CODESYSSPV3/3S/IecVarAccess;String;|var|CODESYS Control Win V3 x64.Application.IOs.SOP710_B1;Write;SOP710_B1;Digital;;
CODESYSSPV3/3S/IecVarAccess;String;|var|CODESYS Control Win V3 x64.Application.IOs.SOP711_FQ1;Write;SOP711_FQ1;Digital;;
CODESYSSPV3/3S/IecVarAccess;String;|var|CODESYS Control Win V3 x64.Application.IOs.SOP711_B1;Write;SOP711_B1;Digital;;
CODESYSSPV3/3S/IecVarAccess;String;|var|CODESYS Control Win V3 x64.Application.IOs.SOP712_FQ1;Write;SOP712_FQ1;Digital;;
CODESYSSPV3/3S/IecVarAccess;String;|var|CODESYS Control Win V3 x64.Application.IOs.SOP712_B1;Write;SOP712_B1;Digital;;
CODESYSSPV3/3S/IecVarAccess;String;|var|CODESYS Control Win V3 x64.Application.IOs.SOP713_FQ1;Write;SOP713_FQ1;Digital;;
CODESYSSPV3/3S/IecVarAccess;String;|var|CODESYS Control Win V3 x64.Application.IOs.SOP713_B1;Write;SOP713_B1;Digital;;
CODESYSSPV3/3S/IecVarAccess;String;|var|CODESYS Control Win V3 x64.Application.IOs.SOP713_B2;Write;SOP713_B2;Digital;;
CODESYSSPV3/3S/IecVarAccess;String;|var|CODESYS Control Win V3 x64.Application.IOs.SOP713_B3;Write;SOP713_B3;Digital;;
CODESYSSPV3/3S/IecVarAccess;String;|var|CODESYS Control Win V3 x64.Application.IOs.SOP714_FQ1;Write;SOP714_FQ1;Digital;;
CODESYSSPV3/3S/IecVarAccess;String;|var|CODESYS Control Win V3 x64.Application.IOs.SOP714_B1;Write;SOP714_B1;Digital;;
CODESYSSPV3/3S/IecVarAccess;String;|var|CODESYS Control Win V3 x64.Application.IOs.SOP715_FQ1;Write;SOP715_FQ1;Digital;;
CODESYSSPV3/3S/IecVarAccess;String;|var|CODESYS Control Win V3 x64.Application.IOs.SOP715_B1;Write;SOP715_B1;Digital;;
CODESYSSPV3/3S/IecVarAccess;String;|var|CODESYS Control Win V3 x64.Application.IOs.SOP716_FQ1;Write;SOP716_FQ1;Digital;;
CODESYSSPV3/3S/IecVarAccess;String;|var|CODESYS Control Win V3 x64.Application.IOs.SOP716_B1;Write;SOP716_B1;Digital;;
CODESYSSPV3/3S/IecVarAccess;String;|var|CODESYS Control Win V3 x64.Application.IOs.SOP717_FQ1;Write;SOP717_FQ1;Digital;;
CODESYSSPV3/3S/IecVarAccess;String;|var|CODESYS Control Win V3 x64.Application.IOs.SOP717_B1;Write;SOP717_B1;Digital;;
CODESYSSPV3/3S/IecVarAccess;String;|var|CODESYS Control Win V3 x64.Application.IOs.SOP720_FQ1;Write;SOP720_FQ1;Digital;;
CODESYSSPV3/3S/IecVarAccess;String;|var|CODESYS Control Win V3 x64.Application.IOs.SOP720_B1;Write;SOP720_B1;Digital;;
CODESYSSPV3/3S/IecVarAccess;String;|var|CODESYS Control Win V3 x64.Application.IOs.SOP720_FQ2;Write;SOP720_FQ2;Digital;;
CODESYSSPV3/3S/IecVarAccess;String;|var|CODESYS Control Win V3 x64.Application.IOs.SOP720_B2;Write;SOP720_B2;Digital;;
CODESYSSPV3/3S/IecVarAccess;String;|var|CODESYS Control Win V3 x64.Application.IOs.SOP720_B3;Write;SOP720_B3;Digital;;
CODESYSSPV3/3S/IecVarAccess;String;|var|CODESYS Control Win V3 x64.Application.IOs.SOP720_LC1_ON;Write;SOP720_LC1_ON;Digital;;
CODESYSSPV3/3S/IecVarAccess;String;|var|CODESYS Control Win V3 x64.Application.IOs.SOP720_LC2_ON;Write;SOP720_LC2_ON;Digital;;
CODESYSSPV3/3S/IecVarAccess;String;|var|CODESYS Control Win V3 x64.Application.IOs.SOP720_B8;Write;SOP720_B8;Digital;;
CODESYSSPV3/3S/IecVarAccess;String;|var|CODESYS Control Win V3 x64.Application.IOs.SOP721_FQ1;Write;SOP721_FQ1;Digital;;
CODESYSSPV3/3S/IecVarAccess;String;|var|CODESYS Control Win V3 x64.Application.IOs.SOP721_B1;Write;SOP721_B1;Digital;;
CODESYSSPV3/3S/IecVarAccess;String;|var|CODESYS Control Win V3 x64.Application.IOs.SOP730_FQ1;Write;SOP730_FQ1;Digital;;
CODESYSSPV3/3S/IecVarAccess;String;|var|CODESYS Control Win V3 x64.Application.IOs.SOP730_B1;Write;SOP730_B1;Digital;;
CODESYSSPV3/3S/IecVarAccess;String;|var|CODESYS Control Win V3 x64.Application.IOs.SOP730_B2;Write;SOP730_B2;Digital;;
CODESYSSPV3/3S/IecVarAccess;String;|var|CODESYS Control Win V3 x64.Application.IOs.SOP730_B3;Write;SOP730_B3;Digital;;
CODESYSSPV3/3S/IecVarAccess;String;|var|CODESYS Control Win V3 x64.Application.IOs.SOP722_FQ1;Write;SOP722_FQ1;Digital;;
CODESYSSPV3/3S/IecVarAccess;String;|var|CODESYS Control Win V3 x64.Application.IOs.SOP722_B1;Write;SOP722_B1;Digital;;
CODESYSSPV3/3S/IecVarAccess;String;|var|CODESYS Control Win V3 x64.Application.IOs.SOP723_FQ1;Write;SOP723_FQ1;Digital;;
CODESYSSPV3/3S/IecVarAccess;String;|var|CODESYS Control Win V3 x64.Application.IOs.SOP723_B1;Write;SOP723_B1;Digital;;
CODESYSSPV3/3S/IecVarAccess;String;|var|CODESYS Control Win V3 x64.Application.IOs.SOP723_LC1_ON;Write;SOP723_LC1_ON;Digital;;
CODESYSSPV3/3S/IecVarAccess;String;|var|CODESYS Control Win V3 x64.Application.IOs.SOP723_LC2_ON;Write;SOP723_LC2_ON;Digital;;
CODESYSSPV3/3S/IecVarAccess;String;|var|CODESYS Control Win V3 x64.Application.IOs.SOP723_B2;Write;SOP723_B2;Digital;;
CODESYSSPV3/3S/IecVarAccess;String;|var|CODESYS Control Win V3 x64.Application.IOs.SOP710_KM1;Read;SOP710_KM1;Digital;;
CODESYSSPV3/3S/IecVarAccess;String;|var|CODESYS Control Win V3 x64.Application.IOs.SOP710_KM2;Read;SOP710_KM2;Digital;;
CODESYSSPV3/3S/IecVarAccess;String;|var|CODESYS Control Win V3 x64.Application.IOs.SOP711_KM1;Read;SOP711_KM1;Digital;;
CODESYSSPV3/3S/IecVarAccess;String;|var|CODESYS Control Win V3 x64.Application.IOs.SOP711_KM2;Read;SOP711_KM2;Digital;;
CODESYSSPV3/3S/IecVarAccess;String;|var|CODESYS Control Win V3 x64.Application.IOs.SOP712_KM1;Read;SOP712_KM1;Digital;;
CODESYSSPV3/3S/IecVarAccess;String;|var|CODESYS Control Win V3 x64.Application.IOs.SOP712_KM2;Read;SOP712_KM2;Digital;;
CODESYSSPV3/3S/IecVarAccess;String;|var|CODESYS Control Win V3 x64.Application.IOs.SOP713_KM1;Read;SOP713_KM1;Digital;;
CODESYSSPV3/3S/IecVarAccess;String;|var|CODESYS Control Win V3 x64.Application.IOs.SOP713_KM2;Read;SOP713_KM2;Digital;;
CODESYSSPV3/3S/IecVarAccess;String;|var|CODESYS Control Win V3 x64.Application.IOs.SOP713_K3;Read;SOP713_K3;Digital;;
CODESYSSPV3/3S/IecVarAccess;String;|var|CODESYS Control Win V3 x64.Application.IOs.SOP713_K4;Read;SOP713_K4;Digital;;
CODESYSSPV3/3S/IecVarAccess;String;|var|CODESYS Control Win V3 x64.Application.IOs.SOP713_K5;Read;SOP713_K5;Digital;;
CODESYSSPV3/3S/IecVarAccess;String;|var|CODESYS Control Win V3 x64.Application.IOs.SOP713_K6;Read;SOP713_K6;Digital;;
CODESYSSPV3/3S/IecVarAccess;String;|var|CODESYS Control Win V3 x64.Application.IOs.SOP714_KM1;Read;SOP714_KM1;Digital;;
CODESYSSPV3/3S/IecVarAccess;String;|var|CODESYS Control Win V3 x64.Application.IOs.SOP714_KM2;Read;SOP714_KM2;Digital;;
CODESYSSPV3/3S/IecVarAccess;String;|var|CODESYS Control Win V3 x64.Application.IOs.SOP715_KM1;Read;SOP715_KM1;Digital;;
CODESYSSPV3/3S/IecVarAccess;String;|var|CODESYS Control Win V3 x64.Application.IOs.SOP715_KM2;Read;SOP715_KM2;Digital;;
CODESYSSPV3/3S/IecVarAccess;String;|var|CODESYS Control Win V3 x64.Application.IOs.SOP716_KM1;Read;SOP716_KM1;Digital;;
CODESYSSPV3/3S/IecVarAccess;String;|var|CODESYS Control Win V3 x64.Application.IOs.SOP716_KM2;Read;SOP716_KM2;Digital;;
CODESYSSPV3/3S/IecVarAccess;String;|var|CODESYS Control Win V3 x64.Application.IOs.SOP717_KM1;Read;SOP717_KM1;Digital;;
CODESYSSPV3/3S/IecVarAccess;String;|var|CODESYS Control Win V3 x64.Application.IOs.SOP717_KM2;Read;SOP717_KM2;Digital;;
CODESYSSPV3/3S/IecVarAccess;String;|var|CODESYS Control Win V3 x64.Application.IOs.SOP720_KM1;Read;SOP720_KM1;Digital;;
CODESYSSPV3/3S/IecVarAccess;String;|var|CODESYS Control Win V3 x64.Application.IOs.SOP720_KM2;Read;SOP720_KM2;Digital;;
CODESYSSPV3/3S/IecVarAccess;String;|var|CODESYS Control Win V3 x64.Application.IOs.SOP720_KM3;Read;SOP720_KM3;Digital;;
CODESYSSPV3/3S/IecVarAccess;String;|var|CODESYS Control Win V3 x64.Application.IOs.SOP720_KM4;Read;SOP720_KM4;Digital;;
CODESYSSPV3/3S/IecVarAccess;String;|var|CODESYS Control Win V3 x64.Application.IOs.SOP720_Pal_Full;Read;SOP720_Pal_Full;Digital;;
CODESYSSPV3/3S/IecVarAccess;String;|var|CODESYS Control Win V3 x64.Application.IOs.SOP720_Pal_Refill;Read;SOP720_Pal_Refill;Digital;;
CODESYSSPV3/3S/IecVarAccess;String;|var|CODESYS Control Win V3 x64.Application.IOs.SOP720_Pal_Dispense;Read;SOP720_Pal_Dispense;Digital;;
CODESYSSPV3/3S/IecVarAccess;String;|var|CODESYS Control Win V3 x64.Application.IOs.SOP721_KM1;Read;SOP721_KM1;Digital;;
CODESYSSPV3/3S/IecVarAccess;String;|var|CODESYS Control Win V3 x64.Application.IOs.SOP721_KM2;Read;SOP721_KM2;Digital;;
CODESYSSPV3/3S/IecVarAccess;String;|var|CODESYS Control Win V3 x64.Application.IOs.SOP730_KM1;Read;SOP730_KM1;Digital;;
CODESYSSPV3/3S/IecVarAccess;String;|var|CODESYS Control Win V3 x64.Application.IOs.SOP730_KM2;Read;SOP730_KM2;Digital;;
CODESYSSPV3/3S/IecVarAccess;String;|var|CODESYS Control Win V3 x64.Application.IOs.SOP730_K2;Read;SOP730_K2;Digital;;
CODESYSSPV3/3S/IecVarAccess;String;|var|CODESYS Control Win V3 x64.Application.IOs.SOP730_K3;Read;SOP730_K3;Digital;;
CODESYSSPV3/3S/IecVarAccess;String;|var|CODESYS Control Win V3 x64.Application.IOs.SOP730_K4;Read;SOP730_K4;Digital;;
CODESYSSPV3/3S/IecVarAccess;String;|var|CODESYS Control Win V3 x64.Application.IOs.SOP730_K5;Read;SOP730_K5;Digital;;
CODESYSSPV3/3S/IecVarAccess;String;|var|CODESYS Control Win V3 x64.Application.IOs.SOP722_KM1;Read;SOP722_KM1;Digital;;
CODESYSSPV3/3S/IecVarAccess;String;|var|CODESYS Control Win V3 x64.Application.IOs.SOP722_KM2;Read;SOP722_KM2;Digital;;
CODESYSSPV3/3S/IecVarAccess;String;|var|CODESYS Control Win V3 x64.Application.IOs.SOP723_KM1;Read;SOP723_KM1;Digital;;
CODESYSSPV3/3S/IecVarAccess;String;|var|CODESYS Control Win V3 x64.Application.IOs.SOP723_KM2;Read;SOP723_KM2;Digital;;
CODESYSSPV3/3S/IecVarAccess;String;|var|CODESYS Control Win V3 x64.Application.IOs.SOP723_K1;Read;SOP723_K1;Digital;;
CODESYSSPV3/3S/IecVarAccess;String;|var|CODESYS Control Win V3 x64.Application.IOs.SOP723_K2;Read;SOP723_K2;Digital;;
CODESYSSPV3/3S/IecVarAccess;String;|var|CODESYS Control Win V3 x64.Application.IOs.SOP740_PickProduct;Read;SOP740_PickProduct;Digital;;
CODESYSSPV3/3S/IecVarAccess;String;|var|CODESYS Control Win V3 x64.Application.IOs.SOP750_K3;Read;SOP750_K3;Digital;;
CODESYSSPV3/3S/IecVarAccess;String;|var|CODESYS Control Win V3 x64.Application.IOs.SOP750_K4;Read;SOP750_K4;Digital;;
CODESYSSPV3/3S/IecVarAccess;String;|var|CODESYS Control Win V3 x64.Application.IOs.SOP750_K5;Read;SOP750_K5;Digital;;
CODESYSSPV3/3S/IecVarAccess;String;|var|CODESYS Control Win V3 x64.Application.IOs.SOP750_K6;Read;SOP750_K6;Digital;;
CODESYSSPV3/3S/IecVarAccess;String;|var|CODESYS Control Win V3 x64.Application.IOs.SOP700_H1;Read;SOP700_H1;Digital;;
CODESYSSPV3/3S/IecVarAccess;String;|var|CODESYS Control Win V3 x64.Application.IOs.SOP700_H4;Read;SOP700_H4;Digital;;
CODESYSSPV3/3S/IecVarAccess;String;|var|CODESYS Control Win V3 x64.Application.IOs.SOP700_H7;Read;SOP700_H7;Digital;;
CODESYSSPV3/3S/IecVarAccess;String;|var|CODESYS Control Win V3 x64.Application.IOs.SOP700_H10;Read;SOP700_H10;Digital;;
CODESYSSPV3/3S/IecVarAccess;String;|var|CODESYS Control Win V3 x64.Application.IOs.SOP700_H11;Read;SOP700_H11;Digital;;
CODESYSSPV3/3S/IecVarAccess;String;|var|CODESYS Control Win V3 x64.Application.IOs.SOP700_H14;Read;SOP700_H14;Digital;;
CODESYSSPV3/3S/IecVarAccess;String;|var|CODESYS Control Win V3 x64.Application.IOs.SOP700_H15;Read;SOP700_H15;Digital;;
CODESYSSPV3/3S/IecVarAccess;String;|var|CODESYS Control Win V3 x64.Application.IOs.SOP700_H16;Read;SOP700_H16;Digital;;
CODESYSSPV3/3S/IecVarAccess;String;|var|CODESYS Control Win V3 x64.Application.IOs.OP60_ProductNr;Write;OP60_ProductNr;Group;;
CODESYSSPV3/3S/IecVarAccess;String;|var|CODESYS Control Win V3 x64.Application.IOs.OP60_IDNumber;Write;OP60_IDNumber;Group;;
CODESYSSPV3/3S/IecVarAccess;String;|var|CODESYS Control Win V3 x64.Application.IOs.Status;Write;Status;Group;;
CODESYSSPV3/3S/IecVarAccess;String;|var|CODESYS Control Win V3 x64.Application.IOs.OP60_B1;Write;OP60_B1;Digital;;
CODESYSSPV3/3S/IecVarAccess;String;|var|CODESYS Control Win V3 x64.Application.IOs.OP60_KM1;Read;OP60_KM1;Digital;;
CODESYSSPV3/3S/IecVarAccess;String;|var|CODESYS Control Win V3 x64.Application.IOs.OP80_B1;Write;OP80_B1;Digital;;
CODESYSSPV3/3S/IecVarAccess;String;|var|CODESYS Control Win V3 x64.Application.IOs.OP80_KM1;Read;OP80_KM1;Digital;;

  - Light Curtain Sensor 1 [smart component] at (-31.6, 0, -77.53) mm
      signals: DI DisableSensor, DO Detection
      connections:
        Light Curtain Sensor 1.DisableSensor -> PlaneSensor.Active
        PlaneSensor.SensorOut -> Light Curtain Sensor 1.Detection
    - PlaneSensor [smart component, from Components\PlaneSensor.rslib] at (2884.52, 14026.71, 333.51) mm, rotated rx 180 ry 0 rz 0 deg
        properties: Origin=[2.28654003266257 4.4307927432671 0.0338898089966275]; Axis1=[2.3 0 0]; Axis2=[0 0 -1.4]; Tag=(none); SensedPart=(none)
      - _sensorPart_ [part], size 2300 x 0 x 1400 mm
  - Light Curtain Sensor 2 [smart component] at (0, -1819.31, 0) mm
      signals: DI DisableSensor, DO Detection
      connections:
        Light Curtain Sensor 2.DisableSensor -> PlaneSensor_2.Active
        PlaneSensor_2.SensorOut -> Light Curtain Sensor 2.Detection
    - PlaneSensor_2 [smart component, from Components\PlaneSensor.rslib] at (0, 0, 396.73) mm
        properties: Origin=[5.139461 9.59591 0.22208]; Axis1=[2.3 0 0]; Axis2=[0 0 1]; Tag=(none); SensedPart=(none)
      - _sensorPart_ [part], size 2300 x 0 x 1000 mm
  - Light Curtain Sensor 3 [smart component] at (0, -6989.64, 0) mm
      signals: DI DisableSensor, DO Detection
      connections:
        Light Curtain Sensor 3.DisableSensor -> PlaneSensor_3.Active
        PlaneSensor_3.SensorOut -> Light Curtain Sensor 3.Detection
    - PlaneSensor_3 [smart component, from Components\PlaneSensor.rslib] at (-89.72, 0, 389.63) mm
        properties: Origin=[5.139461 9.59591 0.22208]; Axis1=[2.4 0 0]; Axis2=[0 0 1]; Tag=(none); SensedPart=(none)
      - _sensorPart_ [part], size 2400 x 0 x 1000 mm
  - Light Curtain Sensor 4 [smart component] at (17259.69, -4413.54, -135.54) mm, rotated rx 0 ry 0 rz 90 deg
      signals: DI DisableSensor, DO Detection
      connections:
        Light Curtain Sensor 4.DisableSensor -> PlaneSensor_4.Active
        PlaneSensor_4.SensorOut -> Light Curtain Sensor 4.Detection
    - PlaneSensor_4 [smart component, from Components\PlaneSensor.rslib] at (-119.79, 209.38, 385.64) mm
        properties: Origin=[5.139461 9.59591 0.22208]; Axis1=[2 0 0]; Axis2=[0 0 1.15]; Tag=(none); SensedPart=(none)
      - _sensorPart_ [part], size 2000 x 0 x 1150 mm
  - Timer [smart component, from Components\Timer.rslib]
      properties: StartTime=0; Interval=0; Repeat=true; CurrentTime=6.648
  - MB16 [part] at (-390.31, 2938.54, 153.88) mm, rotated rx -90 ry 0 rz -174.01 deg, size 307.8 x 156.9 x 705.9 mm
  - MB20 [part] at (-147.63, 1001.42, 153.01) mm, rotated rx 0 ry -90 rz 88.78 deg, size 307.4 x 156.7 x 856 mm
  - MB24 [part] at (0.47, -3.9, 119.32) mm, rotated rx 103.36 ry 0 rz -1.79 deg, size 308.5 x 176.3 x 856.1 mm
  - MB16T [part] at (-61.86, 1998.8, 85.15) mm, rotated rx 57.28 ry 0 rz 90 deg, size 705.9 x 158.8 x 305.9 mm
  - Source [smart component, from Components\Source.rslib]
      properties: Source=MB16; Copy=(none); Parent=(none); Position=[4.025 0.733 1.086]; Orientation=[1.5707963267949 0 0]; Transient=false; PhysicsBehavior=-1
  - Source_2 [smart component, from Components\Source.rslib]
      properties: Source=MB16T; Copy=(none); Parent=(none); Position=[4.025 0.733 1.086]; Orientation=[1.5707963267949 0 1.5707963267949]; Transient=false; PhysicsBehavior=-1
  - Source_3 [smart component, from Components\Source.rslib]
      properties: Source=MB20; Copy=(none); Parent=(none); Position=[4.025 0.733 1.086]; Orientation=[1.5707963267949 0 0]; Transient=false; PhysicsBehavior=-1
  - Source_4 [smart component, from Components\Source.rslib]
      properties: Source=MB24; Copy=(none); Parent=(none); Position=[4.025 0.733 1.086]; Orientation=[1.5707963267949 0 0]; Transient=false; PhysicsBehavior=-1
  - Source_5 [smart component, from Components\Source.rslib]
      properties: Source=EuroPallet (1); Copy=(none); Parent=(none); Position=[6.30744 1.11093 0.60795]; Orientation=[0 0 1.5707963267949]; Transient=false; PhysicsBehavior=-1
  - SOP722 [smart component] at (6333.61, 6970, 616.89) mm, rotated rx 0 ry 0 rz 90 deg
      properties: ForwardSpeed=0.05; ReverseSpeed=-0.05; ConveyorSpeed=0; SpeedForward=0.7; Constant=1E-09; SpeedBackward=-0.6
      signals: DI MotorFWD, DI MotorREV, DO ConveyorError, DI ResetError, DO MotorFeedback, DO BoxSensor
      connections:
        SOP722.MotorFWD -> ?.Enabled
        SOP722.MotorREV -> ?.Enabled
        ?.Output -> ?.Enabled
        SOP722.MotorFWD -> ?.Execute
        SOP722.MotorREV -> ?.Execute
        SOP722.MotorFWD -> ?.A
        SOP722.MotorREV -> ?.B
        ?.Result -> ConveyorSurfaceBehaviour.SurfaceVelocity
        ?.Output -> ConveyorSurfaceBehaviour.SurfaceVelocity
        ?.Output -> ?.InputA
        ?.Output -> ?.InputB
        SOP722.MotorFWD -> ?.InputA
        SOP722.MotorFWD -> ?.InputA
        SOP722.MotorREV -> ?.InputB
        SOP722.MotorFWD -> ?.InputA
        SOP722.MotorFWD -> ?.A
        ?.Result -> ConveyorSurfaceBehaviour.SurfaceVelocity
        SOP722.MotorFWD -> ?.Set
        SOP722.MotorREV -> ?.Set
        SetIdleSpeed.Result -> SetIdleSpeedToConveyor.Execute
        SOP722.MotorFWD -> SetIdleSpeed.A
        SOP722.MotorREV -> SetIdleSpeed.B
        SOP722.MotorFWD -> SetMotorSafetyBreaker.FWD
        SOP722.MotorREV -> SetMotorSafetyBreaker.REV
        ErrorCheckAndBlockingMotorsAndErrorResetLogic.Output -> SetIdleSpeedToConveyor.Execute
        SOP722.ResetError -> ErrorCheckAndBlockingMotorsAndErrorResetLogic.Reset
        SOP722.MotorFWD -> NoErrorAllowFWD.FWD
        ErrorCheckAndBlockingMotorsAndErrorResetLogic.Output -> NoErrorAllowFWD.Error
        NoErrorAllowFWD.Result -> SetForwardSpeedToConveyor.Execute
        SOP722.MotorREV -> NoErrorAllowREV.REV
        ErrorCheckAndBlockingMotorsAndErrorResetLogic.Output -> NoErrorAllowREV.Error
        NoErrorAllowREV.Result -> SetBackwardSpeedToConveyor.Execute
        SetMotorSafetyBreaker.Result -> ErrorCheckAndBlockingMotorsAndErrorResetLogic.Set
        GraphicsHideLogic.Result -> GraphicsHide.Execute
        SOP722.MotorFWD -> GraphicsHideLogic.FWD
        SOP722.MotorREV -> GraphicsHideLogic.REV
        SOP722.MotorFWD -> MotorFeedbackSignalLogic.A
        SOP722.MotorREV -> MotorFeedbackSignalLogic.A
        ErrorCheckAndBlockingMotorsAndErrorResetLogic.Output -> MotorFeedbackSignalLogic.B
        MotorFeedbackSignalLogic.Result -> SOP722.MotorFeedback
        MotorFeedbackSignalLogic.Result -> GraphicsShow.Execute
        ErrorCheckAndBlockingMotorsAndErrorResetLogic.InvOutput -> SOP722.ConveyorError
        SUB100_B1.SensorSignal -> SOP722.BoxSensor
        ?.Result => ?.Count
        ?.Value => ConveyorSurfaceBehaviour.SurfaceVelocity
        ?.Value => ConveyorSurfaceBehaviour.SurfaceVelocity
        ?.Value => ConveyorSurfaceBehaviour.SurfaceVelocity
        ?.Value => ConveyorSurfaceBehaviour.SurfaceVelocity
        ?.Value => ConveyorSurfaceBehaviour.SurfaceVelocity
        ?.Value => ConveyorSurfaceBehaviour.SurfaceVelocity
        SetIdleSpeedToConveyor.Value => ConveyorSurfaceBehaviour.SurfaceVelocity
        SetForwardSpeedToConveyor.Value => ConveyorSurfaceBehaviour.SurfaceVelocity
        SetBackwardSpeedToConveyor.Value => ConveyorSurfaceBehaviour.SurfaceVelocity
        ?.Result => SetForwardSpeedToConveyor.Max
        ?.A => SetBackwardSpeedToConveyor.Min
        ?.Result => SetBackwardSpeedToConveyor.Max
        ?.A => SetForwardSpeedToConveyor.Min
        GraphicsShow.Object => GraphicsHide.Object
        ?.Object => ?.Object
    - ConveyorSurfaceBehaviour [smart component, from Components\PhysicsControl.rslib] at (-850.96, -505.17, -100) mm
        properties: Object=ConveyorSurface; Behavior=2; SurfaceVelocity=2.05049929770199E-14
    - SetIdleSpeedToConveyor [smart component, from Components\Random.rslib] at (-850.96, -505.17, -100) mm
        properties: Value=2.05049929770199E-14; Min=0; Max=1E-13
    - SetBackwardSpeedToConveyor [smart component, from Components\Random.rslib] at (-850.96, -505.17, -100) mm
        properties: Value=-0.69999999999991; Min=-0.7; Max=-0.6999999999999
    - SetForwardSpeedToConveyor [smart component, from Components\Random.rslib] at (-850.96, -505.17, -100) mm
        properties: Value=0.500000000093782; Min=0.5; Max=0.5000000001
    - SetIdleSpeed [smart component, from Components\LogicExpression.rslib] at (-850.96, -505.17, -100) mm
        properties: Expression=not A and not B
    - SetMotorSafetyBreaker [smart component, from Components\LogicExpression.rslib] at (-850.96, -505.17, -100) mm
        properties: Expression=FWD and REV
    - ErrorCheckAndBlockingMotorsAndErrorResetLogic [smart component, from Components\LogicSRLatch.rslib] at (-850.96, -505.17, -100) mm
    - NoErrorAllowFWD [smart component, from Components\LogicExpression.rslib] at (-850.96, -505.17, -100) mm
        properties: Expression=FWD and not Error
    - NoErrorAllowREV [smart component, from Components\LogicExpression.rslib] at (-850.96, -505.17, -100) mm
        properties: Expression=REV and not Error
    - GraphicsShow [smart component, from Components\Show.rslib] at (-850.96, -505.17, -100) mm
        properties: Object=OnOffGfx
    - GraphicsHide [smart component, from Components\Hide.rslib] at (-850.96, -505.17, -100) mm
        properties: Object=OnOffGfx
    - GraphicsHideLogic [smart component, from Components\LogicExpression.rslib] at (-850.96, -505.17, -100) mm
        properties: Expression=not FWD and not REV
    - GraphicsObjects [graphiccomponentgroup] at (-65.23, -0.94, 0) mm, rotated rx 0 ry 0 rz -90 deg
      - OnOffGfx [graphiccomponentgroup] at (514.42, -850.96, -110.92) mm, rotated rx 0 ry 0 rz 90 deg
        - Part_5 [part] at (-19.01, -85.34, -416.89) mm, rotated rx 0 ry 0 rz -90 deg, size 50 x 1701.5 x 100 mm
        - Part_6 [part] at (0, 1062.79, 0) mm, rotated rx 0 ry 0 rz -90 deg, size 50 x 1701.5 x 100 mm
      - ConveyorSurface [part] at (505.17, -850.96, -112.36) mm, rotated rx 0 ry 0 rz 90 deg, size 1712.3 x 1089.6 x 114.1 mm
    - MotorFeedbackSignalLogic [smart component, from Components\LogicExpression.rslib] at (-850.96, -505.17, -100) mm
        properties: Expression=A AND NOT B
    - Conveyor [part] at (-916.73, -600.7, -162.63) mm, rotated rx 0 ry 0 rz 180 deg, size 1700 x 1300 x 500 mm
    - SUB100_B1 [smart component] at (565.82, 599.25, -101.36) mm, rotated rx 0 ry 0 rz 180 deg
        signals: DO SensorSignal
        connections:
          SensorRay.SensorOut -> ?.Active
          ?.Output -> SUB100_B1.SensorSignal
          SensorRay.SensorOut -> LogicGate.InputA
          GraphicSwitch_2.Output -> LogicGate_2.InputA
          LogicGate_2.Output -> LogicGate.InputB
          LogicGate.Output -> SUB100_B1.SensorSignal
      - SensorRay [smart component, from Components\LineSensor.rslib] at (24.04, 61.94, 174.13) mm
          properties: Start=[0 0 0]; End=[5.26116255894493E-07 0.938058416436489 2.90984203399347E-08]; Radius=0.01; SensedPart=(none); SensedPoint=[0 0 0]; Length=0.938058416436637; Tag=(none)
        - _sensorPart_ [part], size 20 x 938.1 x 20 mm
      - SensorMountWorking [part] at (0, 0, 0) mm, size 50 x 50 x 200 mm
      - GraphicSwitch_2 [smart component, from Components\GraphicSwitch.rslib] at (50, 0, 0) mm
          properties: PartHigh=SensorMountBroken; PartLow=SensorMountWorking
      - SensorMountBroken [part] at (0, 0, 0) mm, size 50 x 50 x 200 mm
      - LogicGate [smart component, from Components\LogicGate.rslib]
          properties: Operator=AND; Delay=0
      - LogicGate_2 [smart component, from Components\LogicGate.rslib]
          properties: Operator=NOT; Delay=0
  - SOP723 [smart component] at (6335.13, 8670, 616.89) mm, rotated rx 0 ry 0 rz 90 deg
      properties: ForwardSpeed=0.05; ReverseSpeed=-0.05; ConveyorSpeed=0; SpeedForward=0.7; Constant=1E-09; SpeedBackward=-0.6
      signals: DI MotorFWD, DI MotorREV, DO ConveyorError, DI ResetError, DO MotorFeedback, DO BoxSensor
      connections:
        SOP723.MotorFWD -> ?.Enabled
        SOP723.MotorREV -> ?.Enabled
        ?.Output -> ?.Enabled
        SOP723.MotorFWD -> ?.Execute
        SOP723.MotorREV -> ?.Execute
        SOP723.MotorFWD -> ?.A
        SOP723.MotorREV -> ?.B
        ?.Result -> ConveyorSurfaceBehaviour.SurfaceVelocity
        ?.Output -> ConveyorSurfaceBehaviour.SurfaceVelocity
        ?.Output -> ?.InputA
        ?.Output -> ?.InputB
        SOP723.MotorFWD -> ?.InputA
        SOP723.MotorFWD -> ?.InputA
        SOP723.MotorREV -> ?.InputB
        SOP723.MotorFWD -> ?.InputA
        SOP723.MotorFWD -> ?.A
        ?.Result -> ConveyorSurfaceBehaviour.SurfaceVelocity
        SOP723.MotorFWD -> ?.Set
        SOP723.MotorREV -> ?.Set
        SetIdleSpeed.Result -> SetIdleSpeedToConveyor.Execute
        SOP723.MotorFWD -> SetIdleSpeed.A
        SOP723.MotorREV -> SetIdleSpeed.B
        SOP723.MotorFWD -> SetMotorSafetyBreaker.FWD
        SOP723.MotorREV -> SetMotorSafetyBreaker.REV
        ErrorCheckAndBlockingMotorsAndErrorResetLogic.Output -> SetIdleSpeedToConveyor.Execute
        SOP723.ResetError -> ErrorCheckAndBlockingMotorsAndErrorResetLogic.Reset
        SOP723.MotorFWD -> NoErrorAllowFWD.FWD
        ErrorCheckAndBlockingMotorsAndErrorResetLogic.Output -> NoErrorAllowFWD.Error
        NoErrorAllowFWD.Result -> SetForwardSpeedToConveyor.Execute
        SOP723.MotorREV -> NoErrorAllowREV.REV
        ErrorCheckAndBlockingMotorsAndErrorResetLogic.Output -> NoErrorAllowREV.Error
        NoErrorAllowREV.Result -> SetBackwardSpeedToConveyor.Execute
        SetMotorSafetyBreaker.Result -> ErrorCheckAndBlockingMotorsAndErrorResetLogic.Set
        GraphicsHideLogic.Result -> GraphicsHide.Execute
        SOP723.MotorFWD -> GraphicsHideLogic.FWD
        SOP723.MotorREV -> GraphicsHideLogic.REV
        SOP723.MotorFWD -> MotorFeedbackSignalLogic.A
        SOP723.MotorREV -> MotorFeedbackSignalLogic.A
        ErrorCheckAndBlockingMotorsAndErrorResetLogic.Output -> MotorFeedbackSignalLogic.B
        MotorFeedbackSignalLogic.Result -> SOP723.MotorFeedback
        MotorFeedbackSignalLogic.Result -> GraphicsShow.Execute
        ErrorCheckAndBlockingMotorsAndErrorResetLogic.InvOutput -> SOP723.ConveyorError
        SUB100_B1.SensorSignal -> SOP723.BoxSensor
        ?.Result => ?.Count
        ?.Value => ConveyorSurfaceBehaviour.SurfaceVelocity
        ?.Value => ConveyorSurfaceBehaviour.SurfaceVelocity
        ?.Value => ConveyorSurfaceBehaviour.SurfaceVelocity
        ?.Value => ConveyorSurfaceBehaviour.SurfaceVelocity
        ?.Value => ConveyorSurfaceBehaviour.SurfaceVelocity
        ?.Value => ConveyorSurfaceBehaviour.SurfaceVelocity
        SetIdleSpeedToConveyor.Value => ConveyorSurfaceBehaviour.SurfaceVelocity
        SetForwardSpeedToConveyor.Value => ConveyorSurfaceBehaviour.SurfaceVelocity
        SetBackwardSpeedToConveyor.Value => ConveyorSurfaceBehaviour.SurfaceVelocity
        ?.Result => SetForwardSpeedToConveyor.Max
        ?.A => SetBackwardSpeedToConveyor.Min
        ?.Result => SetBackwardSpeedToConveyor.Max
        ?.A => SetForwardSpeedToConveyor.Min
        GraphicsShow.Object => GraphicsHide.Object
        ?.Object => ?.Object
    - ConveyorSurfaceBehaviour [smart component, from Components\PhysicsControl.rslib] at (-850.96, -505.17, -100) mm
        properties: Object=ConveyorSurface; Behavior=2; SurfaceVelocity=4.58677998491879E-14
    - SetIdleSpeedToConveyor [smart component, from Components\Random.rslib] at (-850.96, -505.17, -100) mm
        properties: Value=4.58677998491879E-14; Min=0; Max=1E-13
    - SetBackwardSpeedToConveyor [smart component, from Components\Random.rslib] at (-850.96, -505.17, -100) mm
        properties: Value=-0.69999999999991; Min=-0.7; Max=-0.6999999999999
    - SetForwardSpeedToConveyor [smart component, from Components\Random.rslib] at (-850.96, -505.17, -100) mm
        properties: Value=0.500000000045699; Min=0.5; Max=0.5000000001
    - SetIdleSpeed [smart component, from Components\LogicExpression.rslib] at (-850.96, -505.17, -100) mm
        properties: Expression=not A and not B
    - SetMotorSafetyBreaker [smart component, from Components\LogicExpression.rslib] at (-850.96, -505.17, -100) mm
        properties: Expression=FWD and REV
    - ErrorCheckAndBlockingMotorsAndErrorResetLogic [smart component, from Components\LogicSRLatch.rslib] at (-850.96, -505.17, -100) mm
    - NoErrorAllowFWD [smart component, from Components\LogicExpression.rslib] at (-850.96, -505.17, -100) mm
        properties: Expression=FWD and not Error
    - NoErrorAllowREV [smart component, from Components\LogicExpression.rslib] at (-850.96, -505.17, -100) mm
        properties: Expression=REV and not Error
    - GraphicsShow [smart component, from Components\Show.rslib] at (-850.96, -505.17, -100) mm
        properties: Object=OnOffGfx
    - GraphicsHide [smart component, from Components\Hide.rslib] at (-850.96, -505.17, -100) mm
        properties: Object=OnOffGfx
    - GraphicsHideLogic [smart component, from Components\LogicExpression.rslib] at (-850.96, -505.17, -100) mm
        properties: Expression=not FWD and not REV
    - GraphicsObjects [graphiccomponentgroup] at (-65.23, -0.94, 0) mm, rotated rx 0 ry 0 rz -90 deg
      - OnOffGfx [graphiccomponentgroup] at (514.42, -850.96, -110.92) mm, rotated rx 0 ry 0 rz 90 deg
        - Part_5 [part] at (-19.01, -85.34, -416.89) mm, rotated rx 0 ry 0 rz -90 deg, size 50 x 1701.5 x 100 mm
        - Part_6 [part] at (0, 1062.79, 0) mm, rotated rx 0 ry 0 rz -90 deg, size 50 x 1701.5 x 100 mm
      - ConveyorSurface [part] at (505.17, -850.96, -112.36) mm, rotated rx 0 ry 0 rz 90 deg, size 1712.3 x 1089.6 x 114.1 mm
    - MotorFeedbackSignalLogic [smart component, from Components\LogicExpression.rslib] at (-850.96, -505.17, -100) mm
        properties: Expression=A AND NOT B
    - Conveyor [part] at (-916.73, -600.7, -162.63) mm, rotated rx 0 ry 0 rz 180 deg, size 1700 x 1300 x 500 mm
    - SUB100_B1 [smart component] at (565.82, 599.25, -101.36) mm, rotated rx 0 ry 0 rz 180 deg
        signals: DO SensorSignal
        connections:
          SensorRay.SensorOut -> ?.Active
          ?.Output -> SUB100_B1.SensorSignal
          SensorRay.SensorOut -> LogicGate.InputA
          GraphicSwitch_2.Output -> LogicGate_2.InputA
          LogicGate_2.Output -> LogicGate.InputB
          LogicGate.Output -> SUB100_B1.SensorSignal
      - SensorRay [smart component, from Components\LineSensor.rslib] at (24.04, 61.94, 174.13) mm
          properties: Start=[0 0 0]; End=[5.26116255894493E-07 0.938058416436489 2.90984203399347E-08]; Radius=0.01; SensedPart=(none); SensedPoint=[0 0 0]; Length=0.938058416436637; Tag=(none)
        - _sensorPart_ [part], size 20 x 938.1 x 20 mm
      - SensorMountWorking [part] at (0, 0, 0) mm, size 50 x 50 x 200 mm
      - GraphicSwitch_2 [smart component, from Components\GraphicSwitch.rslib] at (50, 0, 0) mm
          properties: PartHigh=SensorMountBroken; PartLow=SensorMountWorking
      - SensorMountBroken [part] at (0, 0, 0) mm, size 50 x 50 x 200 mm
      - LogicGate [smart component, from Components\LogicGate.rslib]
          properties: Operator=AND; Delay=0
      - LogicGate_2 [smart component, from Components\LogicGate.rslib]
          properties: Operator=NOT; Delay=0
  - PalletDispensorMovement [smart component]
      signals: DI ReFillPallet, DI Pallet_FilledUp, DI NewPallet
      connections:
        PoseMover_4.Executed -> PoseMover_5.Execute
        PoseMover_6.Executed -> PoseMover_7.Execute
        LogicGate.Output -> PoseMover_3.Execute
        PoseMover_7.Executed -> LogicGate.InputB
        PoseMover_7.Executed -> LogicGate_2.InputB
        LogicGate_2.Output -> PoseMover_3.Execute
        PoseMover_5.Executed -> Timer.Active
        Timer.Output -> PoseMover_6.Execute
        Timer_2.Output -> LogicGate.InputA
        LogicGate.Output -> Timer.Reset
        PalletDispensorMovement.ReFillPallet -> PoseMover_8.Execute
        PalletDispensorMovement.Pallet_FilledUp -> ?.InputA
        PalletDispensorMovement.Pallet_FilledUp -> ?.InputA
        PalletDispensorMovement.Pallet_FilledUp -> PoseMover_3.Execute
        PalletDispensorMovement.NewPallet -> PoseMover_4.Execute
        PalletDispensorMovement.NewPallet -> Timer_2.Active
        PoseMover_5.Executed -> PoseMover_6.Execute
    - PoseMover_3 [smart component, from Components\PoseMover.rslib]
        properties: Mechanism=PalletDispenser; Pose=2; Duration=4
    - PoseMover_4 [smart component, from Components\PoseMover.rslib]
        properties: Mechanism=PalletDispenser; Pose=3; Duration=4
    - PoseMover_5 [smart component, from Components\PoseMover.rslib]
        properties: Mechanism=PalletDispenser; Pose=4; Duration=8
    - PoseMover_6 [smart component, from Components\PoseMover.rslib]
        properties: Mechanism=PalletDispenser; Pose=5; Duration=8
    - PoseMover_7 [smart component, from Components\PoseMover.rslib]
        properties: Mechanism=PalletDispenser; Pose=6; Duration=4
    - PoseMover_8 [smart component, from Components\PoseMover.rslib]
        properties: Mechanism=PalletDispenser; Pose=1; Duration=4
  - PalletDispenser [mechanism] at (0, 0, 0) mm; joint values [0, 0, 0] (rad or m)
      links: Wall, HorizontalBar, LeftClamp, RightClamp
  - EuroPallet (1) [part] at (8313.49, 1114.92, 117.23) mm, rotated rx 0 ry 0 rz 89.94 deg, size 1206.6 x 808.8 x 152.5 mm
  - Buttons [graphiccomponentgroup]
    - FilledPallet [part] at (7471.38, 607.83, 1076.55) mm, rotated rx 0 ry 90 rz 0 deg, size 40 x 39.8 x 10 mm
    - Emergency4 [part] at (7471.38, 607.83, 1236.44) mm, rotated rx 0 ry 90 rz 0 deg, size 40 x 39.8 x 10 mm
    - PalletRemove [part] at (7441.66, 9631.65, 1174.65) mm, rotated rx 0 ry 90 rz 90 deg, size 40 x 39.8 x 10 mm
    - Emergency3 [part] at (7441.66, 9631.65, 1280.76) mm, rotated rx 0 ry 90 rz 90 deg, size 40 x 39.8 x 10 mm
    - Emergency1 [part] at (5192.96, 10430.05, 1449.33) mm, rotated rx 0 ry 90 rz -180 deg, size 40 x 39.8 x 10 mm
    - Emergency2 [part] at (5138.96, 10431.72, 1432.3) mm, rotated rx 0 ry 90 rz -180 deg, size 40 x 39.8 x 10 mm
  - SOP720 [smart component] at (6317, 1700, 617) mm, rotated rx 0 ry 0 rz 90 deg
      properties: ForwardSpeed=0.05; ReverseSpeed=-0.05; ConveyorSpeed=0; SpeedForward=0.7; Constant=1E-09; SpeedBackward=-0.6
      signals: DI MotorFWD, DI MotorREV, DO ConveyorError, DI ResetError, DO MotorFeedback, DI RotateFWD, DI RotateREV, DO RotationFeedback, DO PositionSensorB4, DO PositionSensorB5, DO PositionSensorB6
      connections:
        SetIdleSpeed.Result -> SetIdleSpeedToConveyor.Execute
        SOP720.MotorFWD -> SetIdleSpeed.A
        SOP720.MotorREV -> SetIdleSpeed.B
        SOP720.MotorFWD -> SetMotorSafetyBreaker.FWD
        SOP720.MotorREV -> SetMotorSafetyBreaker.REV
        ErrorCheckAndBlockingMotorsAndErrorResetLogic.Output -> SetIdleSpeedToConveyor.Execute
        SOP720.ResetError -> ErrorCheckAndBlockingMotorsAndErrorResetLogic.Reset
        SOP720.MotorFWD -> NoErrorAllowFWD.FWD
        ErrorCheckAndBlockingMotorsAndErrorResetLogic.Output -> NoErrorAllowFWD.Error
        NoErrorAllowFWD.Result -> SetForwardSpeedToConveyor.Execute
        SOP720.MotorREV -> NoErrorAllowREV.REV
        ErrorCheckAndBlockingMotorsAndErrorResetLogic.Output -> NoErrorAllowREV.Error
        NoErrorAllowREV.Result -> SetBackwardSpeedToConveyor.Execute
        SetMotorSafetyBreaker.Result -> ErrorCheckAndBlockingMotorsAndErrorResetLogic.Set
        GraphicsHideLogic.Result -> GraphicsHide.Execute
        SOP720.MotorFWD -> GraphicsHideLogic.FWD
        SOP720.MotorREV -> GraphicsHideLogic.REV
        SOP720.MotorFWD -> MotorFeedbackSignalLogic.A
        SOP720.MotorREV -> MotorFeedbackSignalLogic.A
        ErrorCheckAndBlockingMotorsAndErrorResetLogic.Output -> MotorFeedbackSignalLogic.B
        MotorFeedbackSignalLogic.Result -> SOP720.MotorFeedback
        MotorFeedbackSignalLogic.Result -> GraphicsShow.Execute
        SOP720.RotateFWD -> ?.Execute
        SOP720.RotateREV -> ?.Execute
        ?.Executing -> SOP720.RotationFeedback
        ?.Executing -> SOP720.RotationFeedback
        ErrorCheckAndBlockingMotorsAndErrorResetLogic.InvOutput -> SOP720.ConveyorError
        SOP720.RotateFWD -> RotatorFWD.Execute
        SOP720.RotateREV -> ?.Execute
        SOP720.RotateREV -> RotatorREV.Execute
        PlaneSensorB4.SensorOut -> SOP720.PositionSensorB4
        PlaneSensorB6.SensorOut -> SOP720.PositionSensorB6
        PlaneSensorB5.SensorOut -> SOP720.PositionSensorB5
        SOP720.RotateFWD -> SOP720.RotationFeedback
        SOP720.RotateREV -> SOP720.RotationFeedback
        SetIdleSpeedToConveyor.Value => ConveyorSurfaceBehaviour.SurfaceVelocity
        SetForwardSpeedToConveyor.Value => ConveyorSurfaceBehaviour.SurfaceVelocity
        SetBackwardSpeedToConveyor.Value => ConveyorSurfaceBehaviour.SurfaceVelocity
        GraphicsShow.Object => GraphicsHide.Object
    - ConveyorSurfaceBehaviour [smart component, from Components\PhysicsControl.rslib] at (-850.96, -505.17, -100) mm
        properties: Object=ConveyorSurface; Behavior=2; SurfaceVelocity=0
    - SetIdleSpeedToConveyor [smart component, from Components\Random.rslib] at (-850.96, -505.17, -100) mm
        properties: Value=0; Min=0; Max=1E-13
    - SetBackwardSpeedToConveyor [smart component, from Components\Random.rslib] at (-850.96, -505.17, -100) mm
        properties: Value=-0.699999999999906; Min=-0.7; Max=-0.6999999999999
    - SetForwardSpeedToConveyor [smart component, from Components\Random.rslib] at (-850.96, -505.17, -100) mm
        properties: Value=0.500000000021327; Min=0.5; Max=0.5000000001
    - SetIdleSpeed [smart component, from Components\LogicExpression.rslib] at (-850.96, -505.17, -100) mm
        properties: Expression=not A and not B
    - SetMotorSafetyBreaker [smart component, from Components\LogicExpression.rslib] at (-850.96, -505.17, -100) mm
        properties: Expression=FWD and REV
    - ErrorCheckAndBlockingMotorsAndErrorResetLogic [smart component, from Components\LogicSRLatch.rslib] at (-850.96, -505.17, -100) mm
    - NoErrorAllowFWD [smart component, from Components\LogicExpression.rslib] at (-850.96, -505.17, -100) mm
        properties: Expression=FWD and not Error
    - NoErrorAllowREV [smart component, from Components\LogicExpression.rslib] at (-850.96, -505.17, -100) mm
        properties: Expression=REV and not Error
    - GraphicsShow [smart component, from Components\Show.rslib] at (-850.96, -505.17, -100) mm
        properties: Object=OnOffGfx
    - GraphicsHide [smart component, from Components\Hide.rslib] at (-850.96, -505.17, -100) mm
        properties: Object=OnOffGfx
    - GraphicsHideLogic [smart component, from Components\LogicExpression.rslib] at (-850.96, -505.17, -100) mm
        properties: Expression=not FWD and not REV
    - GraphicsObjects [graphiccomponentgroup] at (0, 0, -261.68) mm, rotated rx 0 ry 0 rz -91.2 deg
      - OnOffGfx [graphiccomponentgroup] at (515.36, -916.19, 165.2) mm, rotated rx 0 ry 0 rz 90 deg
        - FrameE [part] at (221.83, -88.42, -23.07) mm, size 1370 x 50 x 120 mm
        - FrameB [part] at (221.83, 1063.32, -23.07) mm, size 1370 x 50 x 120 mm
        - FrameC [part] at (1741.48, 853.47, -22.72) mm, rotated rx 0 ry 0 rz 120 deg, size 300 x 50 x 120 mm
        - Frame [part] at (115.23, 829.26, -23.07) mm, rotated rx 0 ry 0 rz 60 deg, size 300 x 50 x 120 mm
        - FrameD [part] at (1741.97, 171.27, 96.95) mm, rotated rx 180 ry 0 rz -120 deg, size 300 x 50 x 120 mm
        - FrameF [part] at (115.25, 195.2, 96.56) mm, rotated rx 180 ry 0 rz -60 deg, size 300 x 50 x 120 mm
      - ConveyorSurface [part] at (506.11, -916.19, 149.32) mm, rotated rx 0 ry 0 rz 90 deg, size 1712.3 x 1089.6 x 114.1 mm
      - 1700x1200x500 [graphiccomponentgroup] at (-645.62, 679.63, -249.56) mm
        - GeneratedPart_49 [part] at (100, -125, 460) mm, rotated rx -90 ry 0 rz -90 deg, size 80 x 80 x 1100 mm
        - GeneratedPart_50 [part] at (100, -250, 460) mm, rotated rx -90 ry 0 rz -90 deg, size 80 x 80 x 1100 mm
        - GeneratedPart_51 [part] at (100, -375, 460) mm, rotated rx -90 ry 0 rz -90 deg, size 80 x 80 x 1100 mm
        - GeneratedPart_52 [part] at (100, -500, 460) mm, rotated rx -90 ry 0 rz -90 deg, size 80 x 80 x 1100 mm
        - GeneratedPart_53 [part] at (100, -625, 460) mm, rotated rx -90 ry 0 rz -90 deg, size 80 x 80 x 1100 mm
        - GeneratedPart_54 [part] at (100, -750, 460) mm, rotated rx -90 ry 0 rz -90 deg, size 80 x 80 x 1100 mm
        - GeneratedPart_55 [part] at (100, -875, 460) mm, rotated rx -90 ry 0 rz -90 deg, size 80 x 80 x 1100 mm
        - GeneratedPart_56 [part] at (100, -1000, 460) mm, rotated rx -90 ry 0 rz -90 deg, size 80 x 80 x 1100 mm
        - GeneratedPart_57 [part] at (100, -1125, 460) mm, rotated rx -90 ry 0 rz -90 deg, size 80 x 80 x 1100 mm
        - GeneratedPart_58 [part] at (100, -1250, 460) mm, rotated rx -90 ry 0 rz -90 deg, size 80 x 80 x 1100 mm
        - RollerE [part] at (403.6, 162.24, 460) mm, rotated rx 90 ry 0 rz 90 deg, size 80 x 78 x 500 mm
        - RollerD [part] at (278.02, 0, 460) mm, rotated rx 90 ry 0 rz 90 deg, size 80 x 80 x 750 mm
        - RollerB [part] at (278.02, -1374.95, 460) mm, rotated rx 90 ry 0 rz 90 deg, size 80 x 80 x 750 mm
        - RollerA [part] at (403.6, -1502.19, 460) mm, rotated rx 90 ry 0 rz 90 deg, size 80 x 78 x 500 mm
        - Frame [part] at (331.73, -1480.59, 380) mm, rotated rx 0 ry 0 rz 150 deg, size 300 x 50 x 120 mm
        - FrameB [part] at (97.67, -1373.99, 380) mm, rotated rx 0 ry 0 rz 90 deg, size 1370 x 50 x 120 mm
        - FrameE [part] at (1249.41, -1373.99, 380) mm, rotated rx 0 ry 0 rz 90 deg, size 1370 x 50 x 120 mm
        - FrameD [part] at (989.72, 146.15, 500.02) mm, rotated rx 180 ry 0 rz -30 deg, size 300 x 50 x 120 mm
        - FrameF [part] at (965.78, -1480.57, 499.63) mm, rotated rx 180 ry 0 rz 30 deg, size 300 x 50 x 120 mm
        - FrameC [part] at (307.52, 145.66, 380.35) mm, rotated rx 0 ry 0 rz -150 deg, size 300 x 50 x 120 mm
      - RotatorPlate [part] at (0, 0, -0.93) mm, rotated rx 0 ry 0 rz 90 deg, size 1600 x 1591.2 x 120 mm
      - SUB200_B1 [smart component] at (-595.62, 542.39, 160.12) mm, rotated rx 0 ry 0 rz -90 deg
          signals: DO SensorSignal
          connections:
            SensorRay.SensorOut -> ?.Active
            ?.Output -> SUB200_B1.SensorSignal
            SensorRay.SensorOut -> SUB200_B1.SensorSignal
        - SensorRay [smart component, from Components\LineSensor.rslib] at (-25.96, 61.94, 174.13) mm
            properties: Start=[0 0 0]; End=[5.96111039252722E-07 0.938058507471307 1.8696271550378E-07]; Radius=0.01; SensedPart=(none); SensedPoint=[0 0 0]; Length=0.938058507471515; Tag=(none)
          - _sensorPart_ [part], size 20 x 938.1 x 20 mm
        - SensorMount [part] at (-50, 0, 0) mm, size 50 x 50 x 200 mm
      - Activator [part] at (0, 490.23, 155.75) mm, rotated rx 0 ry 0 rz 90 deg, size 50 x 10 x 20 mm
    - MotorFeedbackSignalLogic [smart component, from Components\LogicExpression.rslib] at (-850.96, -505.17, -100) mm
        properties: Expression=A AND NOT B
    - RotatorFWD [smart component, from Components\Rotator.rslib]
        properties: Object=GraphicsObjects; CenterPoint=[0 0 0]; Axis=[0 0 1]; Speed=-0.174532925199433; Reference=Local; ReferenceObject=(none)
    - RotatorREV [smart component, from Components\Rotator.rslib]
        properties: Object=GraphicsObjects; CenterPoint=[0 0 0]; Axis=[0 0 1]; Speed=0.174532925199433; Reference=Local; ReferenceObject=(none)
    - PlaneSensorB5 [smart component, from Components\PlaneSensor.rslib] at (-4.28, -534.63, -102.3) mm
        properties: Origin=[0 0 0]; Axis1=[0.005 0 0]; Axis2=[0 0.1 0]; SensedPart=(none); Tag=(none)
      - _sensorPart_ [part], size 5 x 100 x 0 mm
    - PlaneSensorB4 [smart component, from Components\PlaneSensor.rslib] at (534.63, 9.69, -102.3) mm, rotated rx 0 ry 0 rz 90 deg
        properties: Origin=[0 0 0]; Axis1=[0.002 0 0]; Axis2=[0 0.1 0]; SensedPart=(none); Tag=(none)
      - _sensorPart_ [part], size 2 x 100 x 0 mm
    - PlaneSensorB6 [smart component, from Components\PlaneSensor.rslib] at (-13.48, 431.85, -102.3) mm
        properties: Origin=[0 0 0]; Axis1=[0.005 0 0]; Axis2=[0 0.1 0]; SensedPart=(none); Tag=(none)
      - _sensorPart_ [part], size 5 x 100 x 0 mm
    - GFX_legs2 [part] at (410.56, -641.07, -516.89) mm, size 100 x 1300 x 260 mm
    - GFX_legs1 [part] at (-488.8, -641.07, -516.89) mm, size 100 x 1300 x 260 mm
  - SOP730 [smart component] at (6335.96, 5270, 616.89) mm, rotated rx 0 ry 0 rz 90 deg
      properties: ForwardSpeed=0.05; ReverseSpeed=-0.05; ConveyorSpeed=0; SpeedForward=0.7; Constant=1E-09; SpeedBackward=-0.6
      signals: DI MotorFWD, DI MotorREV, DO ConveyorError, DI ResetError, DO MotorFeedback, DI FrontUp, DI FrontDown, DI RearUp, DI RearDown, DO BoxSensor, DO FrontSensor, DO RearSensor
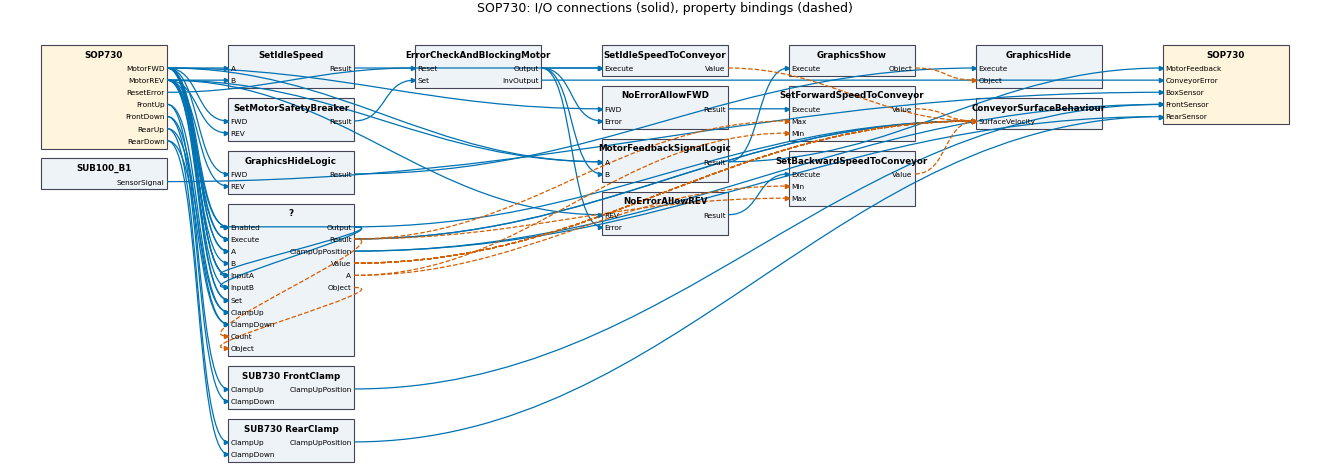
      connections:
        SOP730.MotorFWD -> ?.Enabled
        SOP730.MotorREV -> ?.Enabled
        ?.Output -> ?.Enabled
        SOP730.MotorFWD -> ?.Execute
        SOP730.MotorREV -> ?.Execute
        SOP730.MotorFWD -> ?.A
        SOP730.MotorREV -> ?.B
        ?.Result -> ConveyorSurfaceBehaviour.SurfaceVelocity
        ?.Output -> ConveyorSurfaceBehaviour.SurfaceVelocity
        ?.Output -> ?.InputA
        ?.Output -> ?.InputB
        SOP730.MotorFWD -> ?.InputA
        SOP730.MotorFWD -> ?.InputA
        SOP730.MotorREV -> ?.InputB
        SOP730.MotorFWD -> ?.InputA
        SOP730.MotorFWD -> ?.A
        ?.Result -> ConveyorSurfaceBehaviour.SurfaceVelocity
        SOP730.MotorFWD -> ?.Set
        SOP730.MotorREV -> ?.Set
        SetIdleSpeed.Result -> SetIdleSpeedToConveyor.Execute
        SOP730.MotorFWD -> SetIdleSpeed.A
        SOP730.MotorREV -> SetIdleSpeed.B
        SOP730.MotorFWD -> SetMotorSafetyBreaker.FWD
        SOP730.MotorREV -> SetMotorSafetyBreaker.REV
        ErrorCheckAndBlockingMotorsAndErrorResetLogic.Output -> SetIdleSpeedToConveyor.Execute
        SOP730.ResetError -> ErrorCheckAndBlockingMotorsAndErrorResetLogic.Reset
        SOP730.MotorFWD -> NoErrorAllowFWD.FWD
        ErrorCheckAndBlockingMotorsAndErrorResetLogic.Output -> NoErrorAllowFWD.Error
        NoErrorAllowFWD.Result -> SetForwardSpeedToConveyor.Execute
        SOP730.MotorREV -> NoErrorAllowREV.REV
        ErrorCheckAndBlockingMotorsAndErrorResetLogic.Output -> NoErrorAllowREV.Error
        NoErrorAllowREV.Result -> SetBackwardSpeedToConveyor.Execute
        SetMotorSafetyBreaker.Result -> ErrorCheckAndBlockingMotorsAndErrorResetLogic.Set
        GraphicsHideLogic.Result -> GraphicsHide.Execute
        SOP730.MotorFWD -> GraphicsHideLogic.FWD
        SOP730.MotorREV -> GraphicsHideLogic.REV
        SOP730.MotorFWD -> MotorFeedbackSignalLogic.A
        SOP730.MotorREV -> MotorFeedbackSignalLogic.A
        ErrorCheckAndBlockingMotorsAndErrorResetLogic.Output -> MotorFeedbackSignalLogic.B
        MotorFeedbackSignalLogic.Result -> SOP730.MotorFeedback
        MotorFeedbackSignalLogic.Result -> GraphicsShow.Execute
        ErrorCheckAndBlockingMotorsAndErrorResetLogic.InvOutput -> SOP730.ConveyorError
        SUB100_B1.SensorSignal -> SOP730.BoxSensor
        SUB730 FrontClamp.ClampUpPosition -> SOP730.FrontSensor
        SUB730 RearClamp.ClampUpPosition -> SOP730.RearSensor
        SOP730.FrontUp -> SUB730 FrontClamp.ClampUp
        SOP730.FrontDown -> SUB730 FrontClamp.ClampDown
        SOP730.RearUp -> SUB730 RearClamp.ClampUp
        SOP730.RearDown -> SUB730 RearClamp.ClampDown
        SOP730.FrontUp -> SUB730 FrontClamp.ClampUp
        SOP730.FrontDown -> SUB730 FrontClamp.ClampDown
        SUB730 FrontClamp.ClampUpPosition -> SOP730.FrontSensor
        SOP730.RearUp -> SUB730 RearClamp.ClampUp
        SOP730.RearDown -> SUB730 RearClamp.ClampDown
        SUB730 RearClamp.ClampUpPosition -> SOP730.RearSensor
        ?.Result => ?.Count
        ?.Value => ConveyorSurfaceBehaviour.SurfaceVelocity
        ?.Value => ConveyorSurfaceBehaviour.SurfaceVelocity
        ?.Value => ConveyorSurfaceBehaviour.SurfaceVelocity
        ?.Value => ConveyorSurfaceBehaviour.SurfaceVelocity
        ?.Value => ConveyorSurfaceBehaviour.SurfaceVelocity
        ?.Value => ConveyorSurfaceBehaviour.SurfaceVelocity
        SetIdleSpeedToConveyor.Value => ConveyorSurfaceBehaviour.SurfaceVelocity
        SetForwardSpeedToConveyor.Value => ConveyorSurfaceBehaviour.SurfaceVelocity
        SetBackwardSpeedToConveyor.Value => ConveyorSurfaceBehaviour.SurfaceVelocity
        ?.Result => SetForwardSpeedToConveyor.Max
        ?.A => SetBackwardSpeedToConveyor.Min
        ?.Result => SetBackwardSpeedToConveyor.Max
        ?.A => SetForwardSpeedToConveyor.Min
        GraphicsShow.Object => GraphicsHide.Object
        ?.Object => ?.Object
    - ConveyorSurfaceBehaviour [smart component, from Components\PhysicsControl.rslib] at (-850.96, -505.17, -100) mm
        properties: Object=ConveyorSurface; Behavior=2; SurfaceVelocity=0
    - SetIdleSpeedToConveyor [smart component, from Components\Random.rslib] at (-850.96, -505.17, -100) mm
        properties: Value=0; Min=0; Max=1E-13
    - SetBackwardSpeedToConveyor [smart component, from Components\Random.rslib] at (-850.96, -505.17, -100) mm
        properties: Value=-0.69999999999991; Min=-0.7; Max=-0.6999999999999
    - SetForwardSpeedToConveyor [smart component, from Components\Random.rslib] at (-850.96, -505.17, -100) mm
        properties: Value=0.500000000052467; Min=0.5; Max=0.5000000001
    - SetIdleSpeed [smart component, from Components\LogicExpression.rslib] at (-850.96, -505.17, -100) mm
        properties: Expression=not A and not B
    - SetMotorSafetyBreaker [smart component, from Components\LogicExpression.rslib] at (-850.96, -505.17, -100) mm
        properties: Expression=FWD and REV
    - ErrorCheckAndBlockingMotorsAndErrorResetLogic [smart component, from Components\LogicSRLatch.rslib] at (-850.96, -505.17, -100) mm
    - NoErrorAllowFWD [smart component, from Components\LogicExpression.rslib] at (-850.96, -505.17, -100) mm
        properties: Expression=FWD and not Error
    - NoErrorAllowREV [smart component, from Components\LogicExpression.rslib] at (-850.96, -505.17, -100) mm
        properties: Expression=REV and not Error
    - GraphicsShow [smart component, from Components\Show.rslib] at (-850.96, -505.17, -100) mm
        properties: Object=OnOffGfx
    - GraphicsHide [smart component, from Components\Hide.rslib] at (-850.96, -505.17, -100) mm
        properties: Object=OnOffGfx
    - GraphicsHideLogic [smart component, from Components\LogicExpression.rslib] at (-850.96, -505.17, -100) mm
        properties: Expression=not FWD and not REV
    - GraphicsObjects [graphiccomponentgroup] at (-65.23, -0.94, 0) mm, rotated rx 0 ry 0 rz -90 deg
      - OnOffGfx [graphiccomponentgroup] at (514.42, -850.96, -110.92) mm, rotated rx 0 ry 0 rz 90 deg
        - Part_5 [part] at (-19.01, -85.34, -416.89) mm, rotated rx 0 ry 0 rz -90 deg, size 50 x 1701.5 x 100 mm
        - Part_6 [part] at (0, 1062.79, 0) mm, rotated rx 0 ry 0 rz -90 deg, size 50 x 1701.5 x 100 mm
      - ConveyorSurface [part] at (505.17, -850.96, -112.36) mm, rotated rx 0 ry 0 rz 90 deg, size 1712.3 x 1089.6 x 114.1 mm
    - MotorFeedbackSignalLogic [smart component, from Components\LogicExpression.rslib] at (-850.96, -505.17, -100) mm
        properties: Expression=A AND NOT B
    - Conveyor [part] at (-916.73, -600.7, -162.63) mm, rotated rx 0 ry 0 rz 180 deg, size 1700 x 1300 x 500 mm
    - SUB100_B1 [smart component] at (565.82, 599.25, -101.36) mm, rotated rx 0 ry 0 rz 180 deg
        signals: DO SensorSignal
        connections:
          SensorRay.SensorOut -> ?.Active
          ?.Output -> SUB100_B1.SensorSignal
          SensorRay.SensorOut -> LogicGate.InputA
          GraphicSwitch_2.Output -> LogicGate_2.InputA
          LogicGate_2.Output -> LogicGate.InputB
          LogicGate.Output -> SUB100_B1.SensorSignal
      - SensorRay [smart component, from Components\LineSensor.rslib] at (24.04, 61.94, 174.13) mm
          properties: Start=[0 0 0]; End=[5.26116255894493E-07 0.938058416436489 2.90984203399347E-08]; Radius=0.01; SensedPart=(none); SensedPoint=[0 0 0]; Length=0.938058416436637; Tag=(none)
        - _sensorPart_ [part], size 20 x 938.1 x 20 mm
      - SensorMountWorking [part] at (0, 0, 0) mm, size 50 x 50 x 200 mm
      - GraphicSwitch_2 [smart component, from Components\GraphicSwitch.rslib] at (50, 0, 0) mm
          properties: PartHigh=SensorMountBroken; PartLow=SensorMountWorking
      - SensorMountBroken [part] at (0, 0, 0) mm, size 50 x 50 x 200 mm
      - LogicGate [smart component, from Components\LogicGate.rslib]
          properties: Operator=AND; Delay=0
      - LogicGate_2 [smart component, from Components\LogicGate.rslib]
          properties: Operator=NOT; Delay=0
    - SUB730 FrontClamp [smart component, from Components\SUB730 FrontClamp1.rslib] at (714.35, -108.27, -113.28) mm, rotated rx 0 ry 0 rz 90 deg
        connections:
          SUB730 FrontClamp.ClampUp -> LogicExpression.A
          BottomPosSensor.SensorOut -> LogicExpression.B
          LogicExpression.Result -> LinearMoveUp.Execute
          SUB730 FrontClamp.ClampDown -> LogicExpression_2.A
          BottomPosSensor.SensorOut -> LogicExpression_2.B
          LogicExpression_2.Result -> LinearMoveDown.Execute
          LinearMoveUp.Executed -> LogicSRLatch.Set
          LogicSRLatch.Output -> SUB730 FrontClamp.ClampUpPosition
          LinearMoveDown.Executed -> ?.Set
          ?.Output -> SUB730 FrontClamp.ClampDownPosition
          LinearMoveDown.Executing -> LogicSRLatch.Reset
          LinearMoveUp.Executing -> ?.Reset
          BottomPosSensor.SensorOut -> SUB730 FrontClamp.ClampDownPosition
      - Clamp3D [part, from Components\SUB730 FrontClamp1.rslib]
      - BottomPosSensor [smart component, from Components\LineSensor.rslib] at (18.37, 10.91, 93.4) mm
          properties: Start=[-5.44677247749092E-09 -9.84894448774476E-08 -0.0999997155196143]; End=[-5.44677247749092E-09 -9.84894448774476E-08 -0.0899997155196144]; Radius=0.02; SensedPart=Clamp3D; SensedPoint=[6.425861328125 5.97344140625 0.503608154296875]; Length=0.0099999999999999; Tag=(none)
        - _sensorPart_ [part, from Components\SUB730 FrontClamp1.rslib]
      - LinearMoveUp [smart component, from Components\LinearMover2.rslib]
          properties: Object=Clamp3D; Direction=[0 0 0.1]; Distance=0.1; Duration=1; Reference=Global; ReferenceObject=(none)
      - LinearMoveDown [smart component, from Components\LinearMover2.rslib]
          properties: Object=Clamp3D; Direction=[0 0 -0.1]; Distance=0.1; Duration=1; Reference=Global; ReferenceObject=(none)
      - LogicExpression [smart component, from Components\LogicExpression.rslib]
          properties: Expression=A AND B
      - LogicExpression_2 [smart component, from Components\LogicExpression.rslib]
          properties: Expression=A AND NOT B
      - LogicSRLatch [smart component, from Components\LogicSRLatch.rslib]
    - SUB730 RearClamp [smart component, from Components\SUB730 RearClamp1.rslib] at (-679.81, -100.54, -122.63) mm, rotated rx 0 ry 0 rz 90 deg
        connections:
          SUB730 RearClamp.ClampUp -> LogicExpression.A
          BottomPosSensor.SensorOut -> LogicExpression.B
          LogicExpression.Result -> LinearMoveUp.Execute
          SUB730 RearClamp.ClampDown -> LogicExpression_2.A
          BottomPosSensor.SensorOut -> LogicExpression_2.B
          LogicExpression_2.Result -> LinearMoveDown.Execute
          LinearMoveUp.Executed -> LogicSRLatch.Set
          LogicSRLatch.Output -> SUB730 RearClamp.ClampUpPosition
          LinearMoveDown.Executed -> ?.Set
          ?.Output -> SUB730 RearClamp.ClampDownPosition
          LinearMoveDown.Executing -> LogicSRLatch.Reset
          LinearMoveUp.Executing -> ?.Reset
          BottomPosSensor.SensorOut -> SUB730 RearClamp.ClampDownPosition
      - Clamp3D [part, from Components\SUB730 RearClamp1.rslib]
      - BottomPosSensor [smart component, from Components\LineSensor.rslib] at (18.37, 10.91, 93.4) mm
          properties: Start=[-5.44677247749092E-09 -9.84894448774476E-08 -0.0999997155196143]; End=[-5.44677247749092E-09 -9.84894448774476E-08 -0.0899997155196144]; Radius=0.02; SensedPart=Clamp3D; SensedPoint=[6.41812744140625 4.57928466796875 0.49426123046875]; Length=0.0099999999999999; Tag=(none)
        - _sensorPart_ [part, from Components\SUB730 RearClamp1.rslib]
      - LinearMoveUp [smart component, from Components\LinearMover2.rslib]
          properties: Object=Clamp3D; Direction=[0 0 0.1]; Distance=0.1; Duration=1; Reference=Global; ReferenceObject=(none)
      - LinearMoveDown [smart component, from Components\LinearMover2.rslib]
          properties: Object=Clamp3D; Direction=[0 0 -0.1]; Distance=0.1; Duration=1; Reference=Global; ReferenceObject=(none)
      - LogicExpression [smart component, from Components\LogicExpression.rslib]
          properties: Expression=A AND B
      - LogicExpression_2 [smart component, from Components\LogicExpression.rslib]
          properties: Expression=A AND NOT B
      - LogicSRLatch [smart component, from Components\LogicSRLatch.rslib]
  - Source_6 [smart component, from Components\Source.rslib]
      properties: Source=EuroPallet (1); Copy=(none); Parent=(none); Position=[6.30644 1.11093 0.75195]; Orientation=[0 0 1.5707963267949]; Transient=false; PhysicsBehavior=-1
  - ComponentInstance [part] at (2987197.81, 12313266.11, 3.31) mm, rotated rx 0 ry 0 rz -167.96 deg, size 1206.6 x 808.8 x 152.5 mm
  - SOP721 [smart component] at (6333.61, 3570, 616.89) mm, rotated rx 0 ry 0 rz 90 deg
      properties: ForwardSpeed=0.05; ReverseSpeed=-0.05; ConveyorSpeed=0; SpeedForward=0.7; Constant=1E-09; SpeedBackward=-0.6
      signals: DI MotorFWD, DI MotorREV, DO ConveyorError, DI ResetError, DO MotorFeedback, DO BoxSensor
      connections:
        SOP721.MotorFWD -> ?.Enabled
        SOP721.MotorREV -> ?.Enabled
        ?.Output -> ?.Enabled
        SOP721.MotorFWD -> ?.Execute
        SOP721.MotorREV -> ?.Execute
        SOP721.MotorFWD -> ?.A
        SOP721.MotorREV -> ?.B
        ?.Result -> ConveyorSurfaceBehaviour.SurfaceVelocity
        ?.Output -> ConveyorSurfaceBehaviour.SurfaceVelocity
        ?.Output -> ?.InputA
        ?.Output -> ?.InputB
        SOP721.MotorFWD -> ?.InputA
        SOP721.MotorFWD -> ?.InputA
        SOP721.MotorREV -> ?.InputB
        SOP721.MotorFWD -> ?.InputA
        SOP721.MotorFWD -> ?.A
        ?.Result -> ConveyorSurfaceBehaviour.SurfaceVelocity
        SOP721.MotorFWD -> ?.Set
        SOP721.MotorREV -> ?.Set
        SetIdleSpeed.Result -> SetIdleSpeedToConveyor.Execute
        SOP721.MotorFWD -> SetIdleSpeed.A
        SOP721.MotorREV -> SetIdleSpeed.B
        SOP721.MotorFWD -> SetMotorSafetyBreaker.FWD
        SOP721.MotorREV -> SetMotorSafetyBreaker.REV
        ErrorCheckAndBlockingMotorsAndErrorResetLogic.Output -> SetIdleSpeedToConveyor.Execute
        SOP721.ResetError -> ErrorCheckAndBlockingMotorsAndErrorResetLogic.Reset
        SOP721.MotorFWD -> NoErrorAllowFWD.FWD
        ErrorCheckAndBlockingMotorsAndErrorResetLogic.Output -> NoErrorAllowFWD.Error
        NoErrorAllowFWD.Result -> SetForwardSpeedToConveyor.Execute
        SOP721.MotorREV -> NoErrorAllowREV.REV
        ErrorCheckAndBlockingMotorsAndErrorResetLogic.Output -> NoErrorAllowREV.Error
        NoErrorAllowREV.Result -> SetBackwardSpeedToConveyor.Execute
        SetMotorSafetyBreaker.Result -> ErrorCheckAndBlockingMotorsAndErrorResetLogic.Set
        GraphicsHideLogic.Result -> GraphicsHide.Execute
        SOP721.MotorFWD -> GraphicsHideLogic.FWD
        SOP721.MotorREV -> GraphicsHideLogic.REV
        SOP721.MotorFWD -> MotorFeedbackSignalLogic.A
        SOP721.MotorREV -> MotorFeedbackSignalLogic.A
        ErrorCheckAndBlockingMotorsAndErrorResetLogic.Output -> MotorFeedbackSignalLogic.B
        MotorFeedbackSignalLogic.Result -> SOP721.MotorFeedback
        MotorFeedbackSignalLogic.Result -> GraphicsShow.Execute
        ErrorCheckAndBlockingMotorsAndErrorResetLogic.InvOutput -> SOP721.ConveyorError
        SUB100_B1.SensorSignal -> SOP721.BoxSensor
        ?.Result => ?.Count
        ?.Value => ConveyorSurfaceBehaviour.SurfaceVelocity
        ?.Value => ConveyorSurfaceBehaviour.SurfaceVelocity
        ?.Value => ConveyorSurfaceBehaviour.SurfaceVelocity
        ?.Value => ConveyorSurfaceBehaviour.SurfaceVelocity
        ?.Value => ConveyorSurfaceBehaviour.SurfaceVelocity
        ?.Value => ConveyorSurfaceBehaviour.SurfaceVelocity
        SetIdleSpeedToConveyor.Value => ConveyorSurfaceBehaviour.SurfaceVelocity
        SetForwardSpeedToConveyor.Value => ConveyorSurfaceBehaviour.SurfaceVelocity
        SetBackwardSpeedToConveyor.Value => ConveyorSurfaceBehaviour.SurfaceVelocity
        ?.Result => SetForwardSpeedToConveyor.Max
        ?.A => SetBackwardSpeedToConveyor.Min
        ?.Result => SetBackwardSpeedToConveyor.Max
        ?.A => SetForwardSpeedToConveyor.Min
        GraphicsShow.Object => GraphicsHide.Object
        ?.Object => ?.Object
    - ConveyorSurfaceBehaviour [smart component, from Components\PhysicsControl.rslib] at (-850.96, -505.17, -100) mm
        properties: Object=ConveyorSurface; Behavior=2; SurfaceVelocity=8.97274357218889E-14
    - SetIdleSpeedToConveyor [smart component, from Components\Random.rslib] at (-850.96, -505.17, -100) mm
        properties: Value=8.97274357218889E-14; Min=0; Max=1E-13
    - SetBackwardSpeedToConveyor [smart component, from Components\Random.rslib] at (-850.96, -505.17, -100) mm
        properties: Value=-0.69999999999991; Min=-0.7; Max=-0.6999999999999
    - SetForwardSpeedToConveyor [smart component, from Components\Random.rslib] at (-850.96, -505.17, -100) mm
        properties: Value=0.500000000079187; Min=0.5; Max=0.5000000001
    - SetIdleSpeed [smart component, from Components\LogicExpression.rslib] at (-850.96, -505.17, -100) mm
        properties: Expression=not A and not B
    - SetMotorSafetyBreaker [smart component, from Components\LogicExpression.rslib] at (-850.96, -505.17, -100) mm
        properties: Expression=FWD and REV
    - ErrorCheckAndBlockingMotorsAndErrorResetLogic [smart component, from Components\LogicSRLatch.rslib] at (-850.96, -505.17, -100) mm
    - NoErrorAllowFWD [smart component, from Components\LogicExpression.rslib] at (-850.96, -505.17, -100) mm
        properties: Expression=FWD and not Error
    - NoErrorAllowREV [smart component, from Components\LogicExpression.rslib] at (-850.96, -505.17, -100) mm
        properties: Expression=REV and not Error
    - GraphicsShow [smart component, from Components\Show.rslib] at (-850.96, -505.17, -100) mm
        properties: Object=OnOffGfx
    - GraphicsHide [smart component, from Components\Hide.rslib] at (-850.96, -505.17, -100) mm
        properties: Object=OnOffGfx
    - GraphicsHideLogic [smart component, from Components\LogicExpression.rslib] at (-850.96, -505.17, -100) mm
        properties: Expression=not FWD and not REV
    - GraphicsObjects [graphiccomponentgroup] at (-65.23, -0.94, 0) mm, rotated rx 0 ry 0 rz -90 deg
      - OnOffGfx [graphiccomponentgroup] at (514.42, -850.96, -110.92) mm, rotated rx 0 ry 0 rz 90 deg
        - Part_5 [part] at (-19.01, -85.34, -416.89) mm, rotated rx 0 ry 0 rz -90 deg, size 50 x 1701.5 x 100 mm
        - Part_6 [part] at (0, 1062.79, 0) mm, rotated rx 0 ry 0 rz -90 deg, size 50 x 1701.5 x 100 mm
      - ConveyorSurface [part] at (505.17, -850.96, -112.36) mm, rotated rx 0 ry 0 rz 90 deg, size 1712.3 x 1089.6 x 114.1 mm
    - MotorFeedbackSignalLogic [smart component, from Components\LogicExpression.rslib] at (-850.96, -505.17, -100) mm
        properties: Expression=A AND NOT B
    - Conveyor [part] at (-916.73, -600.7, -162.63) mm, rotated rx 0 ry 0 rz 180 deg, size 1700 x 1300 x 500 mm
    - SUB100_B1 [smart component] at (565.82, 599.25, -101.36) mm, rotated rx 0 ry 0 rz 180 deg
        signals: DO SensorSignal
        connections:
          SensorRay.SensorOut -> ?.Active
          ?.Output -> SUB100_B1.SensorSignal
          SensorRay.SensorOut -> LogicGate.InputA
          GraphicSwitch_2.Output -> LogicGate_2.InputA
          LogicGate_2.Output -> LogicGate.InputB
          LogicGate.Output -> SUB100_B1.SensorSignal
      - SensorRay [smart component, from Components\LineSensor.rslib] at (24.04, 61.94, 174.13) mm
          properties: Start=[0 0 0]; End=[5.26116255894493E-07 0.938058416436489 2.90984203399347E-08]; Radius=0.01; SensedPart=(none); SensedPoint=[0 0 0]; Length=0.938058416436637; Tag=(none)
        - _sensorPart_ [part], size 20 x 938.1 x 20 mm
      - SensorMountWorking [part] at (0, 0, 0) mm, size 50 x 50 x 200 mm
      - GraphicSwitch_2 [smart component, from Components\GraphicSwitch.rslib] at (50, 0, 0) mm
          properties: PartHigh=SensorMountBroken; PartLow=SensorMountWorking
      - SensorMountBroken [part] at (0, 0, 0) mm, size 50 x 50 x 200 mm
      - LogicGate [smart component, from Components\LogicGate.rslib]
          properties: Operator=AND; Delay=0
      - LogicGate_2 [smart component, from Components\LogicGate.rslib]
          properties: Operator=NOT; Delay=0
Station signals: DI NewMB16, DI NewMB16T, DI NewMB20, DI NewMB24, DI NewPallet
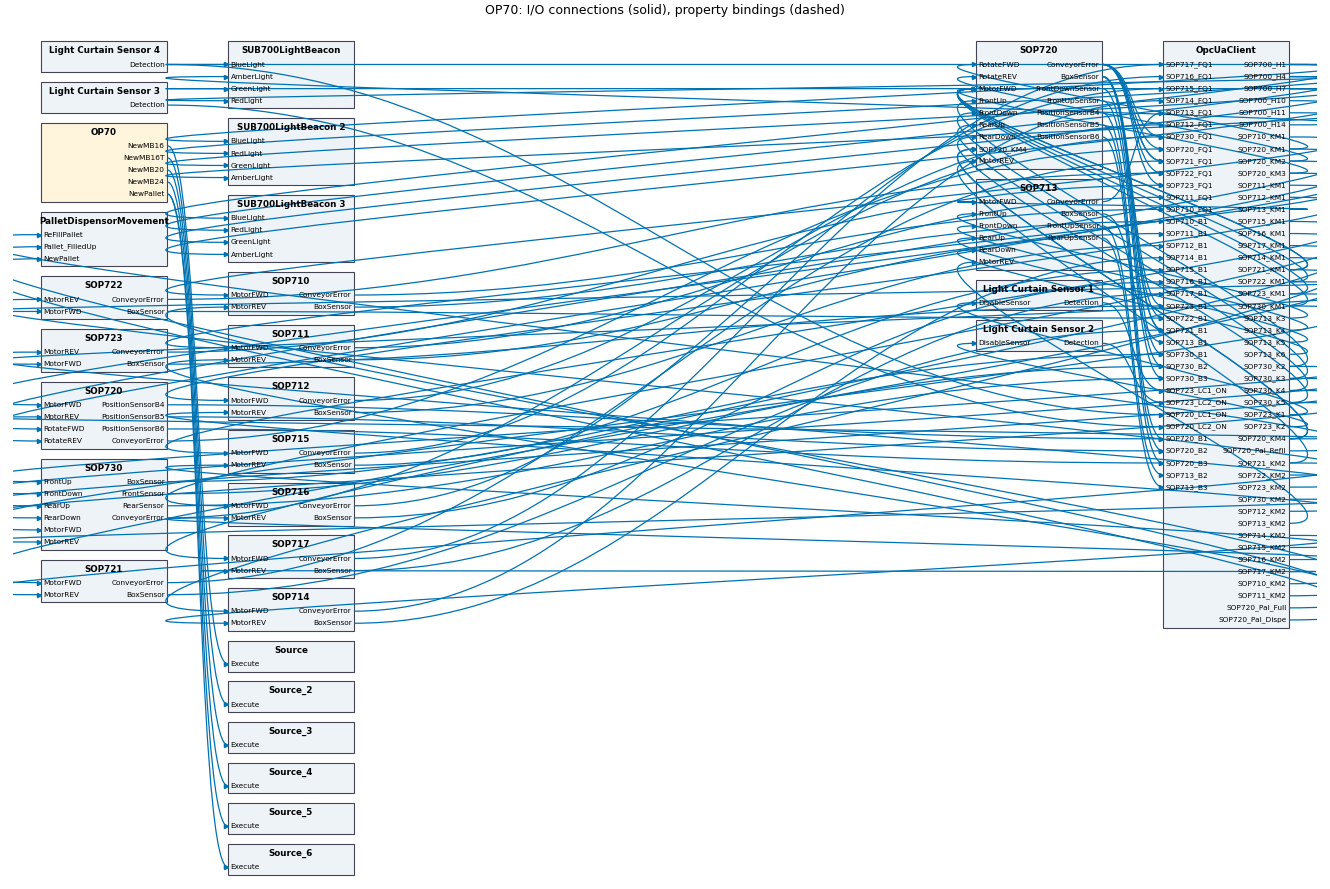
Station logic (signal -> signal, property => property):
  OpcUaClient.SOP700_H1 -> SUB700LightBeacon.BlueLight
  OpcUaClient.SOP700_H1 -> SUB700LightBeacon 2.BlueLight
  OpcUaClient.SOP700_H1 -> SUB700LightBeacon 3.BlueLight
  OpcUaClient.SOP700_H4 -> SUB700LightBeacon 2.RedLight
  OpcUaClient.SOP700_H4 -> SUB700LightBeacon 3.RedLight
  OpcUaClient.SOP700_H7 -> SUB700LightBeacon 2.GreenLight
  OpcUaClient.SOP700_H7 -> SUB700LightBeacon 3.GreenLight
  OpcUaClient.SOP700_H10 -> SUB700LightBeacon 3.AmberLight
  OpcUaClient.SOP700_H11 -> SUB700LightBeacon 2.AmberLight
  OpcUaClient.SOP700_H14 -> SUB700LightBeacon.AmberLight
  OpcUaClient.SOP710_KM1 -> SOP710.MotorFWD
  OpcUaClient.SOP720_KM1 -> SOP720.RotateFWD
  OpcUaClient.SOP720_KM2 -> SOP720.RotateREV
  OpcUaClient.SOP720_KM3 -> SOP720.MotorFWD
  OpcUaClient.SOP711_KM1 -> SOP711.MotorFWD
  OpcUaClient.SOP712_KM1 -> SOP712.MotorFWD
  OpcUaClient.SOP713_KM1 -> SOP713.MotorFWD
  OpcUaClient.SOP715_KM1 -> SOP715.MotorFWD
  OpcUaClient.SOP716_KM1 -> SOP716.MotorFWD
  OpcUaClient.SOP717_KM1 -> SOP717.MotorFWD
  OpcUaClient.SOP714_KM1 -> SOP714.MotorFWD
  SOP717.ConveyorError -> OpcUaClient.SOP717_FQ1
  SOP716.ConveyorError -> OpcUaClient.SOP716_FQ1
  SOP715.ConveyorError -> OpcUaClient.SOP715_FQ1
  SOP714.ConveyorError -> OpcUaClient.SOP714_FQ1
  SOP713.ConveyorError -> OpcUaClient.SOP713_FQ1
  SOP712.ConveyorError -> OpcUaClient.SOP712_FQ1
  SOP730.ConveyorError -> OpcUaClient.SOP730_FQ1
  SOP720.ConveyorError -> OpcUaClient.SOP720_FQ1
  SOP721.ConveyorError -> OpcUaClient.SOP721_FQ1
  SOP722.ConveyorError -> OpcUaClient.SOP722_FQ1
  SOP723.ConveyorError -> OpcUaClient.SOP723_FQ1
  OpcUaClient.SOP721_KM1 -> SOP721.MotorFWD
  OpcUaClient.SOP722_KM1 -> SOP722.MotorFWD
  OpcUaClient.SOP723_KM1 -> SOP723.MotorFWD
  OpcUaClient.SOP730_KM1 -> SOP730.MotorFWD
  SOP711.ConveyorError -> OpcUaClient.SOP711_FQ1
  SOP710.ConveyorError -> OpcUaClient.SOP710_FQ1
  SOP710.BoxSensor -> OpcUaClient.SOP710_B1
  SOP711.BoxSensor -> OpcUaClient.SOP711_B1
  SOP712.BoxSensor -> OpcUaClient.SOP712_B1
  SOP714.BoxSensor -> OpcUaClient.SOP714_B1
  SOP715.BoxSensor -> OpcUaClient.SOP715_B1
  SOP716.BoxSensor -> OpcUaClient.SOP716_B1
  SOP717.BoxSensor -> OpcUaClient.SOP717_B1
  SOP723.BoxSensor -> OpcUaClient.SOP723_B1
  SOP722.BoxSensor -> OpcUaClient.SOP722_B1
  SOP721.BoxSensor -> OpcUaClient.SOP721_B1
  SOP713.BoxSensor -> OpcUaClient.SOP713_B1
  OpcUaClient.SOP713_K3 -> SOP713.FrontUp
  OpcUaClient.SOP713_K4 -> SOP713.FrontDown
  OpcUaClient.SOP713_K5 -> SOP713.RearUp
  OpcUaClient.SOP713_K6 -> SOP713.RearDown
  SOP730.BoxSensor -> OpcUaClient.SOP730_B1
  SOP730.FrontDownSensor -> OpcUaClient.SOP730_B2
  SOP730.FrontUpSensor -> OpcUaClient.SOP730_B3
  OpcUaClient.SOP730_K2 -> SOP730.FrontUp
  OpcUaClient.SOP730_K3 -> SOP730.FrontDown
  OpcUaClient.SOP730_K4 -> SOP730.RearUp
  OpcUaClient.SOP730_K5 -> SOP730.RearDown
  OpcUaClient.SOP723_K1 -> Light Curtain Sensor 1.DisableSensor
  OpcUaClient.SOP723_K2 -> Light Curtain Sensor 2.DisableSensor
  Light Curtain Sensor 1.Detection -> OpcUaClient.SOP723_LC1_ON
  Light Curtain Sensor 2.Detection -> OpcUaClient.SOP723_LC2_ON
  Light Curtain Sensor 4.Detection -> OpcUaClient.SOP720_LC1_ON
  Light Curtain Sensor 3.Detection -> OpcUaClient.SOP720_LC2_ON
  OpcUaClient.SOP720_KM4 -> Pallet Dispenser Movement Right.SOP720_KM4
  OpcUaClient.SOP720_KM4 -> Pallet Dispenser Movement Left.SOP720_KM4
  SOP720.PositionSensorB4 -> OpcUaClient.SOP720_B1
  SOP720.PositionSensorB5 -> OpcUaClient.SOP720_B2
  SOP720.PositionSensorB6 -> OpcUaClient.SOP720_B3
  OP70.NewMB16 -> Source.Execute
  OP70.NewMB16T -> Source_2.Execute
  OP70.NewMB20 -> Source_3.Execute
  OP70.NewMB24 -> Source_4.Execute
  OP70.NewPallet -> Source_5.Execute
  SOP713.FrontUpSensor -> OpcUaClient.SOP713_B2
  SOP713.RearUpSensor -> OpcUaClient.SOP713_B3
  OpcUaClient.SOP720_Pal_Refill -> PalletDispensorMovement.ReFillPallet
  SOP721.ConveyorError -> OpcUaClient.SOP721_FQ1
  SOP721.BoxSensor -> OpcUaClient.SOP721_B1
  SOP722.ConveyorError -> OpcUaClient.SOP722_FQ1
  SOP722.BoxSensor -> OpcUaClient.SOP722_B1
  SOP723.ConveyorError -> OpcUaClient.SOP723_FQ1
  SOP723.BoxSensor -> OpcUaClient.SOP723_B1
  OpcUaClient.SOP721_KM2 -> SOP721.MotorREV
  OpcUaClient.SOP722_KM2 -> SOP722.MotorREV
  OpcUaClient.SOP723_KM2 -> SOP723.MotorREV
  OpcUaClient.SOP721_KM1 -> SOP721.MotorFWD
  OpcUaClient.SOP722_KM1 -> SOP722.MotorFWD
  OpcUaClient.SOP723_KM1 -> SOP723.MotorFWD
  SOP720.PositionSensorB4 -> OpcUaClient.SOP720_B1
  SOP720.PositionSensorB5 -> OpcUaClient.SOP720_B2
  SOP720.PositionSensorB6 -> OpcUaClient.SOP720_B3
  OpcUaClient.SOP720_KM3 -> SOP720.MotorFWD
  OpcUaClient.SOP720_KM4 -> SOP720.MotorREV
  OpcUaClient.SOP720_KM1 -> SOP720.RotateFWD
  OpcUaClient.SOP720_KM2 -> SOP720.RotateREV
  SOP730.BoxSensor -> OpcUaClient.SOP730_B1
  SOP730.FrontSensor -> OpcUaClient.SOP730_B2
  SOP730.RearSensor -> OpcUaClient.SOP730_B3
  OpcUaClient.SOP730_K2 -> SOP730.FrontUp
  OpcUaClient.SOP730_K3 -> SOP730.FrontDown
  OpcUaClient.SOP730_K4 -> SOP730.RearUp
  OpcUaClient.SOP730_K5 -> SOP730.RearDown
  OpcUaClient.SOP730_KM1 -> SOP730.MotorFWD
  OpcUaClient.SOP730_KM2 -> SOP730.MotorREV
  SOP730.ConveyorError -> OpcUaClient.SOP730_FQ1
  SOP720.ConveyorError -> OpcUaClient.SOP720_FQ1
  OpcUaClient.SOP700_H7 -> SUB700LightBeacon.GreenLight
  OpcUaClient.SOP700_H4 -> SUB700LightBeacon.RedLight
  OpcUaClient.SOP712_KM2 -> SOP712.MotorREV
  OpcUaClient.SOP713_KM2 -> SOP713.MotorREV
  OpcUaClient.SOP714_KM2 -> SOP714.MotorREV
  OpcUaClient.SOP715_KM2 -> SOP715.MotorREV
  OpcUaClient.SOP716_KM2 -> SOP716.MotorREV
  OpcUaClient.SOP717_KM2 -> SOP717.MotorREV
  OpcUaClient.SOP710_KM2 -> SOP710.MotorREV
  OpcUaClient.SOP711_KM2 -> SOP711.MotorREV
  OP70.NewPallet -> Source_6.Execute
  OpcUaClient.SOP720_Pal_Full -> PalletDispensorMovement.Pallet_FilledUp
  OpcUaClient.SOP720_Pal_Dispense -> PalletDispensorMovement.NewPallet
  SOP721.ConveyorError -> OpcUaClient.SOP721_FQ1
  SOP721.BoxSensor -> OpcUaClient.SOP721_B1
  OpcUaClient.SOP721_KM1 -> SOP721.MotorFWD
  OpcUaClient.SOP721_KM2 -> SOP721.MotorREV
